# EPICS autosave request: sscanApp/Db/scanProgress_settings.req
$(P)hangWaitSec
